PROGRAM Analyzers
VAR
	PM_beck_EL3453:			FB_EL3453_handling;
	
	S_nom_facility_inv:			REAL; //Inverse of Snom [1/kVA]
	V_nom_facility_inv:			REAL; //Inverse of Snom [1/V]
END_VAR

VAR CONSTANT
	tick_hourly: 				REAL:= 2.78E-7; //ms expressed in hours (how much hours is a tick)
END_VAR


PM_beck_EL3453(Analyzer_str_out=> GVL_POWERMETER.Power_analyzer);

//Per unit values obtention - Single-phase powers
GVL_POWERMETER.Power_analyzer.P_L1_pu:= GVL_POWERMETER.Power_analyzer.P_L1_kW * S_nom_facility_inv;
GVL_POWERMETER.Power_analyzer.P_L2_pu:= GVL_POWERMETER.Power_analyzer.P_L2_kW * S_nom_facility_inv;
GVL_POWERMETER.Power_analyzer.P_L3_pu:= GVL_POWERMETER.Power_analyzer.P_L3_kW * S_nom_facility_inv;
GVL_POWERMETER.Power_analyzer.Q_L1_pu:= GVL_POWERMETER.Power_analyzer.Q_L1_kVAr * S_nom_facility_inv;
GVL_POWERMETER.Power_analyzer.Q_L2_pu:= GVL_POWERMETER.Power_analyzer.Q_L2_kVAr * S_nom_facility_inv;
GVL_POWERMETER.Power_analyzer.Q_L3_pu:= GVL_POWERMETER.Power_analyzer.Q_L3_kVAr * S_nom_facility_inv;
GVL_POWERMETER.Power_analyzer.S_L1_pu:= GVL_POWERMETER.Power_analyzer.S_L1_kVA * S_nom_facility_inv;
GVL_POWERMETER.Power_analyzer.S_L2_pu:= GVL_POWERMETER.Power_analyzer.S_L2_kVA * S_nom_facility_inv;
GVL_POWERMETER.Power_analyzer.S_L3_pu:= GVL_POWERMETER.Power_analyzer.S_L3_kVA * S_nom_facility_inv;

//Per unit values obtention - Three-phase powers
GVL_POWERMETER.Power_analyzer.P_pu:= GVL_POWERMETER.Power_analyzer.P_kW * S_nom_facility_inv;
GVL_POWERMETER.Power_analyzer.Q_pu:= GVL_POWERMETER.Power_analyzer.Q_kVAr * S_nom_facility_inv;
GVL_POWERMETER.Power_analyzer.S_pu:= GVL_POWERMETER.Power_analyzer.S_kVA * S_nom_facility_inv;

//Per unit values obtention - Voltages
GVL_POWERMETER.Power_analyzer.V_line_avg_pu:= GVL_POWERMETER.Power_analyzer.V_line_avg_Volt * V_nom_facility_inv;
GVL_POWERMETER.Power_analyzer.V_phase_avg_pu:= GVL_POWERMETER.Power_analyzer.V_phase_avg_Volt * V_nom_facility_inv;

//Active energies calculation. It is an infinitesimal addition (an integration of P_measured)
GVL_POWERMETER.Power_analyzer.Active_er_tot_kWh:= REAL_TO_LINT(GVL_POWERMETER.Power_analyzer.P_kW * tick_hourly) + 
												GVL_POWERMETER.Power_analyzer.Active_er_tot_kWh;
IF GVL_POWERMETER.Power_analyzer.P_kW  >= 0 THEN
	GVL_POWERMETER.Power_analyzer.Active_er_pos_kWh:= REAL_TO_LINT(GVL_POWERMETER.Power_analyzer.P_kW * tick_hourly) + 
													GVL_POWERMETER.Power_analyzer.Active_er_pos_kWh;
ELSE	
	GVL_POWERMETER.Power_analyzer.Active_er_neg_kWh:= REAL_TO_LINT(GVL_POWERMETER.Power_analyzer.P_kW * tick_hourly) + 
													GVL_POWERMETER.Power_analyzer.Active_er_neg_kWh;
END_IF
	
//Reactive energies calculation. It is an infinitesimal addition (an integration of Q_measured)
GVL_POWERMETER.Power_analyzer.React_er_tot_kVArh:= REAL_TO_LINT(GVL_POWERMETER.Power_analyzer.Q_kVAr * tick_hourly) + 
												GVL_POWERMETER.Power_analyzer.React_er_tot_kVArh;
IF GVL_POWERMETER.Power_analyzer.Q_kVAr >= 0 THEN
	GVL_POWERMETER.Power_analyzer.React_er_pos_kVArh:= REAL_TO_LINT(GVL_POWERMETER.Power_analyzer.Q_kVAr * tick_hourly) + 
													GVL_POWERMETER.Power_analyzer.React_er_pos_kVArh;
ELSE
	GVL_POWERMETER.Power_analyzer.React_er_neg_kVArh:= REAL_TO_LINT(GVL_POWERMETER.Power_analyzer.Q_kVAr * tick_hourly) + 
													GVL_POWERMETER.Power_analyzer.React_er_neg_kVArh;
END_IF

//Energies reset when desired
IF GVL_POWERMETER.Energies_reset THEN
	GVL_POWERMETER.Power_analyzer.Active_er_neg_kWh:= 0;
	GVL_POWERMETER.Power_analyzer.Active_er_pos_kWh:= 0;
	GVL_POWERMETER.Power_analyzer.Active_er_tot_kWh:= 0;
	GVL_POWERMETER.Power_analyzer.React_er_neg_kVArh:= 0;
	GVL_POWERMETER.Power_analyzer.React_er_pos_kVArh:= 0;
	GVL_POWERMETER.Power_analyzer.React_er_tot_kVArh:= 0;
	
	GVL_POWERMETER.Energies_reset:= FALSE;
END_IF

END_PROGRAM

(* stored: Version 1.1.0.1, ProductVersion 3.1.4024.11
   POU Analyzers: Id {907aa627-47e3-4482-a979-79b393bfe7d2}, SpecialFunc None *)
